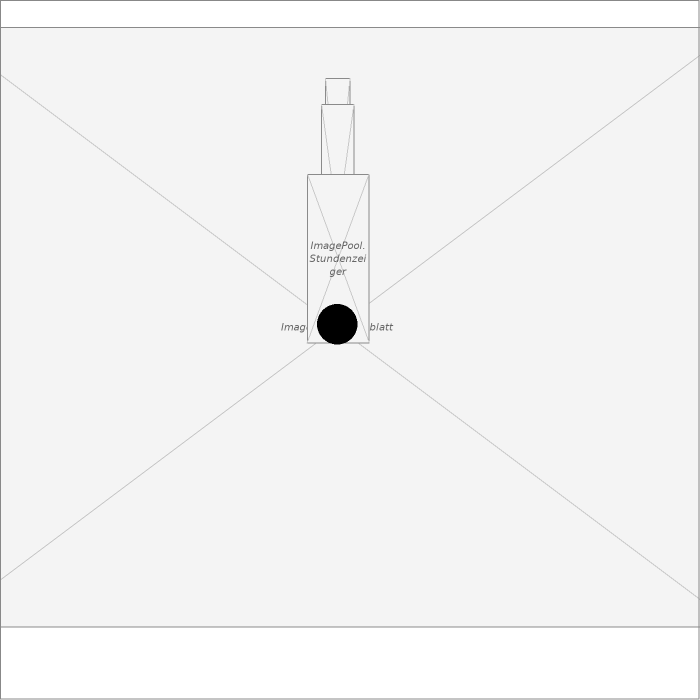
VISUALIZATION Uhr  // 700x700
    Image (-63,27 800x600), image: ImagePool.Ziffernblatt
    Image (325,78 25x260), image: ImagePool.Sekundenzeiger
        p2858320360: Uhr.Sekunde
    Image (321,104 33x239), image: ImagePool.Minutenzeiger
        p2858320360: Uhr.Minute
    Image (307,174 62x169), image: ImagePool.Stundenzeiger
        p2858320360: Uhr.Stunde
    Ellipse (317,304 40x40)
END_VISUALIZATION

(* stored: Version 1.1.0.1, ProductVersion 3.1.4018.5
   Visu Uhr: Id {48cc837c-bc72-481a-8d09-0dd20239bb55} *)
